// TwinCAT 3 PLC project Main
// ProgramVersion: 3.1.4023.0
// libraries:
//   Tc2_Standard, * (Beckhoff Automation GmbH)
//   Tc2_System, * (Beckhoff Automation GmbH)
//   Tc3_Module, * (Beckhoff Automation GmbH)
// project tree:
//   DUTs/ MyStructure.TcDUT
//   GVLs/ GVL.TcGVL
//   / PlcTask.TcTTO (not stored)
//   POUs/ MAIN.TcPOU (not stored)
// real-time tasks:
//   TASK PlcTask: cycle T#10ms, priority 20, ADS port 350

// ---- DUTs/MyStructure.TcDUT
TYPE MyStructure :
STRUCT
	Name : STRING;
	Age : INT;
END_STRUCT
END_TYPE

// ---- GVLs/GVL.TcGVL
{attribute 'qualified_only'}
VAR_GLOBAL
	myArray : ARRAY [0..2] OF MyStructure;
END_VAR
